% RSLogix 500 project GAME SHOW.RSS, saved by version 8.30.00.16 %
PROJECT "UNTITLED"    % processor: MicroLogix 1000 %

PROGRAM FILES
  LAD 2 "MAIN_PROG"  8 rungs
  LAD 3 "COUNTER"  4 rungs
  LAD 4 "FLASHER"  5 rungs
  LAD 5 "STI_INT"  1 rungs
  LAD 6, 7, 8, 9, 10, 11, 12, 13, 14, 15, 16: only END

DATA FILES
  O0 OUTPUT  1 elements
  I1 INPUT  2 elements
  S2 STATUS  33 elements
  B3 BINARY  32 elements
  T4 TIMER  40 elements
  C5 COUNTER  32 elements
  R6 CONTROL  16 elements
  N7 INTEGER  105 elements

LADDER 2 "MAIN_PROG"
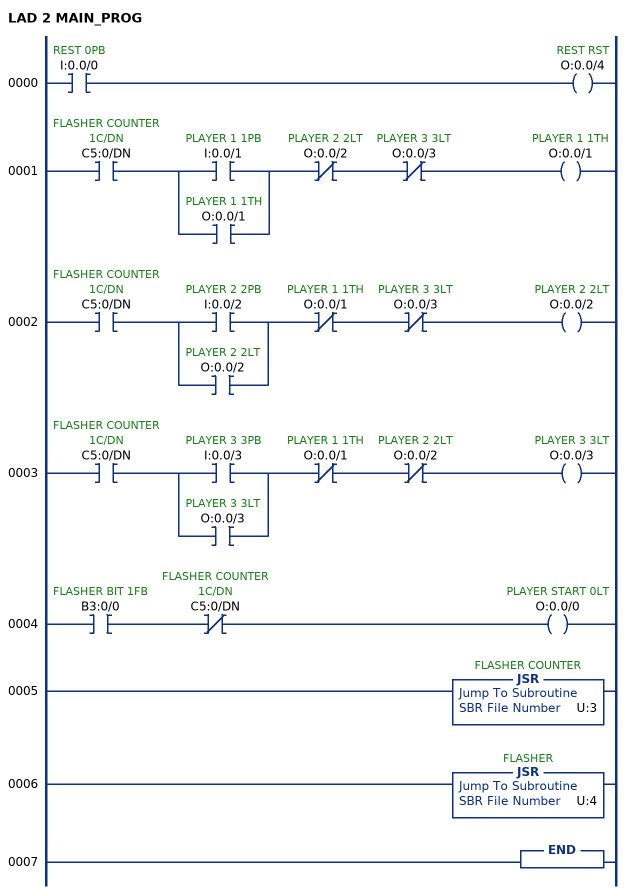
% Rung: 0 %
SOR XIC I:0.0/0 OTE O:0.0/4 EOR
%   I:0.0/0  0PB  "REST" %
%   O:0.0/4  RST  "REST" %
% Rung: 1 %
SOR XIC C5:0/DN BST XIC I:0.0/1 NXB XIC O:0.0/1 BND XIO O:0.0/2 XIO O:0.0/3 OTE O:0.0/1 EOR
%   C5:0  1C  "FLASHER COUNTER" %
%   I:0.0/1  1PB  "PLAYER 1" %
%   O:0.0/1  1TH  "PLAYER 1" %
%   O:0.0/2  2LT  "PLAYER 2" %
%   O:0.0/3  3LT  "PLAYER 3" %
% Rung: 2 %
SOR XIC C5:0/DN BST XIC I:0.0/2 NXB XIC O:0.0/2 BND XIO O:0.0/1 XIO O:0.0/3 OTE O:0.0/2 EOR
%   C5:0  1C  "FLASHER COUNTER" %
%   I:0.0/2  2PB  "PLAYER 2" %
%   O:0.0/2  2LT  "PLAYER 2" %
%   O:0.0/1  1TH  "PLAYER 1" %
%   O:0.0/3  3LT  "PLAYER 3" %
% Rung: 3 %
SOR XIC C5:0/DN BST XIC I:0.0/3 NXB XIC O:0.0/3 BND XIO O:0.0/1 XIO O:0.0/2 OTE O:0.0/3 EOR
%   C5:0  1C  "FLASHER COUNTER" %
%   I:0.0/3  3PB  "PLAYER 3" %
%   O:0.0/3  3LT  "PLAYER 3" %
%   O:0.0/1  1TH  "PLAYER 1" %
%   O:0.0/2  2LT  "PLAYER 2" %
% Rung: 4 %
SOR XIC B3:0/0 XIO C5:0/DN OTE O:0.0/0 EOR
%   B3:0/0  1FB  "FLASHER BIT" %
%   C5:0  1C  "FLASHER COUNTER" %
%   O:0.0/0  0LT  "PLAYER START" %
% Rung: 5 %
SOR JSR U:3 EOR
%   U:3  "FLASHER COUNTER" %
% Rung: 6 %
SOR JSR U:4 EOR
%   U:4  "FLASHER" %
% Rung: 7 %
SOR END EOR

LADDER 3 "COUNTER"
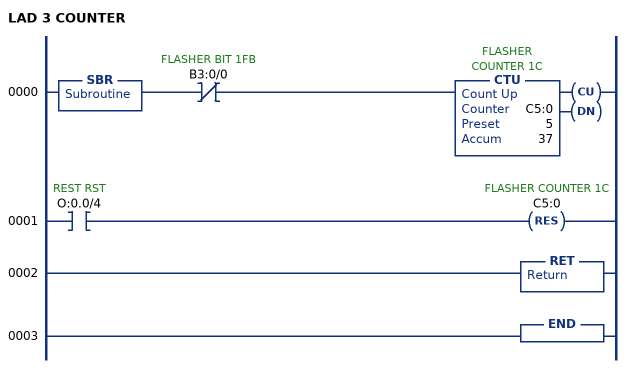
% Rung: 0 %
SOR SBR XIO B3:0/0 CTU C5:0 5 37 EOR
%   B3:0/0  1FB  "FLASHER BIT" %
%   C5:0  1C  "FLASHER COUNTER" %
% Rung: 1 %
SOR XIC O:0.0/4 RES C5:0 EOR
%   O:0.0/4  RST  "REST" %
%   C5:0  1C  "FLASHER COUNTER" %
% Rung: 2 %
SOR RET EOR
% Rung: 3 %
SOR END EOR

LADDER 4 "FLASHER"
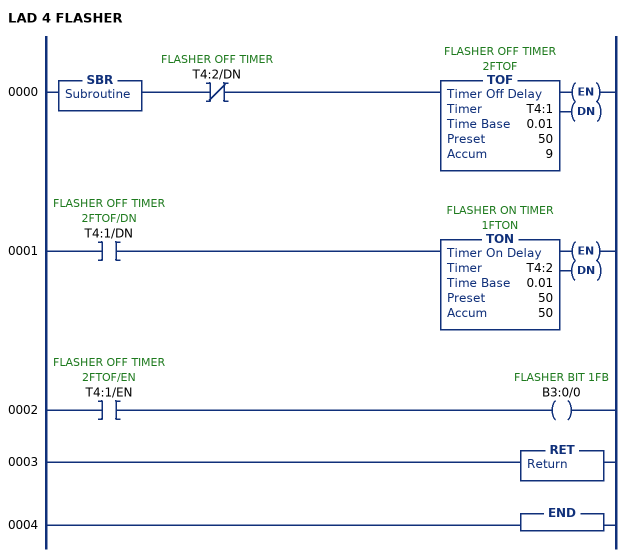
% Rung: 0 %
SOR SBR XIO T4:2/DN TOF T4:1 0.01 50 9 EOR
%   T4:2/DN  "FLASHER OFF TIMER" %
%   T4:1  2FTOF  "FLASHER OFF TIMER" %
% Rung: 1 %
SOR XIC T4:1/DN TON T4:2 0.01 50 50 EOR
%   T4:1  2FTOF  "FLASHER OFF TIMER" %
%   T4:2  1FTON  "FLASHER ON TIMER" %
% Rung: 2 %
SOR XIC T4:1/EN OTE B3:0/0 EOR
%   T4:1  2FTOF  "FLASHER OFF TIMER" %
%   B3:0/0  1FB  "FLASHER BIT" %
% Rung: 3 %
SOR RET EOR
% Rung: 4 %
SOR END EOR

OTHER DOCUMENTED ADDRESSES
  B3  
  B3:0/1  BR1  "PLAYER 1"
  B3:0/2  BR2  "PLAYER 2"
  B3:0/3  BR3  "PLAYER 3"
  B3:0/4  BT4  "PLAYER 1"
  B3:0/5  BT5  "PLAYER 2"
  B3:0/6  BT6  "PLAYER 3"
  B3:0/7  BT7  "PLAYER 1"
  B3:0/8  BT8  "PLAYER 2"
  B3:0/9  BT_9  "PLAYER 3"
  B30:0/1  1BT  "PLAYER 1"
  B30:0/2  BT2  "PLAYER 2"
  B30:0/3  BT3  "PLAYER 3"
  O:0.0/5  "RESET STOP"

DATA TABLE (non-zero values as saved)
DATA B3
% B3:0 % 0X0001 0X0000 0X0000 0X0000 0X0000 0X0000 0X0000 0X0000 0X0000 0X0000
DATA T4
% .PRE .ACC %
% T4:1 % 50 9
% T4:2 % 50 50
DATA C5
% .PRE .ACC %
% C5:0 % 5 37
